Yaskawa INFORM job: X2_34-37(-90,0).JBI

/JOB
//NAME X2_34-37(-90,0)
//POS
///NPOS 361,361,361,9,0,0
///TOOL 0
///POSTYPE PULSE
///PULSE
C00000=-109615,-71844,-36862,18422,13388,2271
C00001=-107008,40287,15446,7646,74688,11911
C00002=-107149,45804,24218,7788,72161,11701
C00003=-108392,48192,28010,10243,72680,1076
C00004=-108392,48392,29954,10302,71604,983
C00005=-108392,48331,29423,10286,71896,1009
C00006=-108010,50265,31522,10186,71551,1114
C00007=-108392,48331,29423,10286,71896,1009
C00008=-108911,49901,30550,10443,72076,8021
C00009=-109414,51873,32709,10619,71831,7821
C00010=-108911,49901,30550,10443,72076,8021
C00011=-102203,43615,23227,8248,72569,10434
C00012=-106081,49085,29485,15378,74997,2308
C00013=-106081,49206,30588,15419,74401,2232
C00014=-106081,49153,30130,15402,74647,2263
C00015=-105730,50968,32108,15326,74307,2347
C00016=-106081,49153,30130,15402,74647,2263
C00017=-108167,43461,21271,12324,74506,6920
C00018=-107374,42085,15448,7738,75637,11845
C00019=-120191,30165,1303,6226,81332,-6626
C00020=-119709,34887,8992,6124,79003,-6581
C00021=-119523,36874,12198,6088,78043,-6565
C00022=-119519,36825,13807,6108,77033,-6613
C00023=-119523,36874,12198,6088,78043,-6565
C00024=-119515,36764,13496,6103,77191,-6604
C00025=-119868,39633,16467,6214,76866,-6741
C00026=-119515,36764,13496,6103,77191,-6604
C00027=-121889,32783,9008,6775,78090,-7366
C00028=-122776,40716,17165,7052,77228,-7717
C00029=-121823,41691,18182,6780,77023,-7402
C00030=-122776,40716,17165,7052,77228,-7717
C00031=-121889,32783,9008,6775,78090,-7366
C00032=-119523,36874,12198,6088,78043,-6565
C00033=-119709,34887,8992,6124,79003,-6581
C00034=-120191,30165,1303,6226,81332,-6626
C00035=-121604,30205,1144,6630,81559,-7083
C00036=-121089,34887,8794,6520,79231,-7034
C00037=-120890,36858,11983,6481,78271,-7017
C00038=-120886,36803,13585,6502,77262,-7069
C00039=-120890,36858,11983,6481,78271,-7017
C00040=-120878,36774,13282,6496,77432,-7057
C00041=-121214,39658,16269,6601,77105,-7189
C00042=-120878,36774,13282,6496,77432,-7057
C00043=-120486,37076,13561,6383,77385,-6926
C00044=-119528,38122,14634,6107,77190,-6608
C00045=-120486,37076,13561,6383,77385,-6926
C00046=-120682,35058,10322,6419,78351,-6942
C00047=-121186,30266,2562,6523,80690,-6990
C00048=-134026,40869,15057,-4047,52311,-47824
C00049=-133273,45805,23219,-4742,49872,-47398
C00050=-132981,47914,26662,-5033,48858,-47219
C00051=-132978,48047,28467,-5116,47820,-47163
C00052=-132981,47914,26662,-5033,48858,-47219
C00053=-132969,48064,28169,-5108,48012,-47169
C00054=-133143,51303,31704,-5016,47492,-47220
C00055=-132969,48064,28169,-5108,48012,-47169
C00056=-135543,46606,26609,-3148,48091,-48321
C00057=-135868,54135,34684,-2953,46980,-48432
C00058=-134925,54643,35244,-3684,46935,-48001
C00059=-135868,54135,34684,-2953,46980,-48432
C00060=-135543,46606,26609,-3148,48091,-48321
C00061=-132981,47914,26662,-5033,48858,-47219
C00062=-133273,45805,23219,-4742,49872,-47398
C00063=-134026,40869,15057,-4047,52311,-47824
C00064=-158164,35728,9631,12841,54320,-57618
C00065=-156933,39530,16487,12369,51918,-57402
C00066=-156452,41160,19364,12190,50934,-57317
C00067=-156450,41229,21096,12367,49926,-57444
C00068=-156452,41160,19364,12190,50934,-57317
C00069=-156479,41102,20610,12346,50159,-57426
C00070=-156356,44237,23924,12335,49721,-57428
C00071=-156479,41102,20610,12346,50159,-57426
C00072=-155785,40986,20547,11858,50036,-57137
C00073=-154785,40646,20189,11137,49940,-56708
C00074=-155785,40986,20547,11858,50036,-57137
C00075=-156262,39303,17617,12037,51024,-57224
C00076=-157483,35375,10637,12509,53434,-57446
C00077=-160593,39475,13550,14508,54241,-58615
C00078=-159342,43270,20469,14089,51785,-58436
C00079=-158853,44905,23381,13934,50776,-58367
C00080=-158852,45007,25149,14138,49770,-58512
C00081=-158853,44905,23381,13934,50776,-58367
C00082=-158854,44932,24718,14094,49990,-58481
C00083=-158703,48121,28150,14084,49505,-58485
C00084=-158854,44932,24718,14094,49990,-58481
C00085=-161444,46441,26342,15939,50249,-59595
C00086=-161040,53766,34331,15923,49060,-59612
C00087=-160097,53171,33669,15238,48978,-59196
C00088=-161040,53766,34331,15923,49060,-59612
C00089=-161444,46441,26342,15939,50249,-59595
C00090=-158853,44905,23381,13934,50776,-58367
C00091=-159342,43270,20469,14089,51785,-58436
C00092=-160593,39475,13550,14508,54241,-58615
C00093=-148971,42504,16746,4915,52183,-53021
C00094=-147979,47046,24523,4355,49683,-52716
C00095=-147593,48996,27807,4132,48646,-52593
C00096=-147590,49137,29621,4197,47605,-52637
C00097=-147593,48996,27807,4132,48646,-52593
C00098=-147610,49163,29309,4198,47810,-52637
C00099=-147661,52475,32942,4273,47281,-52683
C00100=-147610,49163,29309,4198,47810,-52637
C00101=-147454,49128,29272,4080,47808,-52567
C00102=-147457,49325,29466,4083,47790,-52569
C00103=-146486,49526,29681,3347,47716,-52137
C00104=-147457,49325,29466,4083,47790,-52569
C00105=-147454,49128,29272,4080,47808,-52567
C00106=-147593,48996,27807,4132,48646,-52593
C00107=-147979,47046,24523,4355,49683,-52716
C00108=-148753,37651,9035,4624,54413,-52827
C00109=-169007,70240,20067,15770,96475,-54777
C00110=-175404,86334,34832,19373,106938,-55773
C00111=-174173,83341,34513,19133,105400,-55601
C00112=-180960,60737,17059,33421,95392,-55152
C00113=-182232,58952,17300,36312,92073,-55823
C00114=-179527,69319,26237,30671,91177,-56324
C00115=-179117,69620,25739,29739,90864,-56355
C00116=-180097,67994,26330,32410,86483,-57198
C00117=-174100,64042,14056,17976,91926,-56289
C00118=-175447,65123,11808,18399,94042,-56406
C00119=-164161,72,-39985,-6764,90046,-34295
C00120=-130432,-55243,-47386,-13424,82603,8412
C00121=-110572,-56965,-55890,-14658,90278,14468
C00122=-134387,-39172,-38807,12376,86277,-20344
C00123=-136266,-41846,-34601,16059,78566,-27361
C00124=-135424,-39022,-31748,15965,78109,-27121
C00125=-132144,-43884,-34748,15569,76844,-26110
C00126=-133349,-52476,-37829,19150,70304,-22714
C00127=-132707,-53219,-38228,19044,70026,-22517
C00128=-133874,-49344,-36092,21066,73724,-26553
C00129=-127403,-56601,-39797,20204,70737,-24655
C00130=-130575,-58808,-42172,20683,71834,-25657
C00131=-131419,-52897,-41760,13173,72105,-2236
C00132=-151757,-37235,-32664,25855,92713,-16023
C00133=-148694,-31120,-30848,28555,97484,-16481
C00134=-152363,20888,-11521,23566,108052,-25705
C00135=-155491,63274,13853,18429,111086,-34801
C00136=-150514,89045,46229,21307,107758,-32982
C00137=-149106,88504,48693,21100,105732,-32842
C00138=-153882,51041,13508,33623,93530,-12210
C00139=-152694,62068,23397,30426,96150,-11386
C00140=-153686,72545,35966,30292,92124,-9774
C00141=-151360,57639,18849,26215,86885,985
C00142=-146574,44978,5250,17386,80629,11620
C00143=-146389,46654,5686,14273,81867,14897
C00144=-140559,38264,-1160,881,75419,28460
C00145=-140619,46287,2526,1728,82676,28626
C00146=-139837,43342,-3801,1439,85041,28899
C00147=-141798,27002,-27786,2149,91441,28405
C00148=-143772,-19107,-38740,14355,94017,-12677
C00149=-143698,-35148,-33847,20276,92427,-33189
C00150=-141918,-24797,-26817,20326,92921,-32464
C00151=-139594,-23350,-22642,20301,90627,-32011
C00152=-140432,-46735,-33066,23878,71822,-30909
C00153=-143639,-38419,-27501,28411,78321,-12621
C00154=-143508,-41209,-28848,28005,73462,-10092
C00155=-137835,-52557,-35170,23319,62427,898
C00156=-129144,-60406,-38739,13300,52691,14440
C00157=-124267,-62455,-40002,3057,50573,24449
C00158=-118897,-58306,-39599,-7322,55586,36992
C00159=-117935,-60108,-42034,-7672,56240,37337
C00160=-115664,-65010,-47736,-8512,57449,38158
C00161=-121785,-61828,-52329,-5505,69210,35118
C00162=-148930,-33628,-41038,4538,77484,18447
C00163=-163858,24222,1645,10794,81228,7547
C00164=-163712,28964,9442,10824,78886,7392
C00165=-163498,30748,12887,10810,77675,7358
C00166=-163094,25533,8827,6495,74182,-305
C00167=-171402,35198,19720,19438,77476,-19020
C00168=-175083,69400,56807,24741,86302,-36577
C00169=-176478,62304,51821,30230,71876,-61965
C00170=-174700,53660,39403,25265,70725,-61619
C00171=-176244,52382,34806,25393,73168,-61673
C00172=-174832,57379,31343,14926,87681,-59388
C00173=-147451,1111,-29714,5377,100632,-19781
C00174=-112791,-31989,-50015,-2241,90212,24459
C00175=-107981,-35875,-46971,-4517,78040,26268
C00176=-109410,-31915,-41181,-4141,76439,25836
C00177=-109671,-29943,-38250,-4081,75635,25773
C00178=-108634,-25346,-36028,-8315,81190,19632
C00179=-113738,-28838,-38579,-3049,79626,8435
C00180=-120146,-28716,-38356,4151,79685,-1679
C00181=-136605,-12769,-23758,24735,88388,-21929
C00182=-138977,-10728,-20961,25939,84821,-23296
C00183=-136358,-19206,-27135,20431,74888,-32424
C00184=-127631,-24253,-35023,5775,74490,-30240
C00185=-129181,-27934,-40726,6212,76213,-30690
C00186=-139651,-3107,-33687,4364,86662,15844
C00187=-140099,618,-27389,4493,84729,15631
C00188=-140095,1958,-24533,4497,83662,15594
C00189=-138507,5371,-22539,-1336,86874,9491
C00190=-148370,2023,-23416,11466,83880,-10285
C00191=-153111,8749,-17173,17827,86768,-20413
C00192=-156427,18095,-8041,22706,89820,-28931
C00193=-159438,37588,11995,27333,93831,-28775
C00194=-154226,15962,-9104,16757,78816,-38782
C00195=-152712,20066,-9195,12847,84122,-38020
C00196=-154297,18366,-13942,13242,86364,-38311
C00197=-143466,6998,19042,5158,32162,-41222
C00198=-147237,-51968,-50099,-4175,73083,-42408
C00199=3643,-76224,-106676,19950,71810,76872
C00200=6047,-95755,-92046,-14751,98253,9605
C00201=8024,-164446,-133802,-16041,6272,12396
C00202=8024,-164446,-133802,-16041,6272,12396
C00203=80911,-131071,-112390,-19160,57527,-4768
C00204=107387,-112645,-89313,-18613,48039,-3448
C00205=120529,-94925,-67119,-18087,38914,-2179
C00206=102807,-11704,-32462,-5874,76695,-13415
C00207=103436,-3791,-23255,-6127,75148,-13126
C00208=103560,-1765,-20423,-6188,74460,-13051
C00209=103560,-1806,-19122,-6212,73642,-13010
C00210=103601,-1431,-19452,-6214,74041,-13015
C00211=104452,277,-18031,-6506,74110,-12725
C00212=103539,-2063,-20212,-6189,74177,-13043
C00213=120126,-10436,-31938,-6011,80471,6680
C00214=119034,-8056,-29018,-5697,79822,6345
C00215=119034,-8150,-28117,-5707,79221,6375
C00216=119034,-8056,-29018,-5697,79822,6345
C00217=118636,-7203,-28340,-5579,79816,6211
C00218=119064,-5644,-27091,-5704,79877,6351
C00219=118636,-7203,-28340,-5579,79816,6211
C00220=122253,-9472,-30321,-6643,80135,7408
C00221=122707,-3013,-24427,-6779,79866,7571
C00222=122021,-2022,-23613,-6578,79819,7343
C00223=122707,-3013,-24427,-6779,79866,7571
C00224=121204,9301,-16198,-6319,81003,7011
C00225=120979,11415,-12534,-6272,79823,6996
C00226=120979,11346,-11871,-6278,79382,7018
C00227=120979,11415,-12534,-6272,79823,6996
C00228=121673,13624,-10544,-6477,79786,7230
C00229=120979,11415,-12534,-6272,79823,6996
C00230=121039,12182,-11846,-8037,80321,9006
C00231=120294,13253,-10880,-7825,80206,8763
C00232=121039,12182,-11846,-8037,80321,9006
C00233=121310,5674,-20943,-6336,82061,6993
C00234=139815,-25323,-43479,-19,53677,50237
C00235=137572,-18164,-33682,1617,51348,49297
C00236=137572,-18186,-32944,1627,50884,49290
C00237=137572,-18164,-33682,1617,51348,49297
C00238=138000,-16627,-32540,1306,51428,49477
C00239=137572,-18164,-33682,1617,51348,49297
C00240=141541,-18207,-34048,-1274,51544,50959
C00241=141186,-12326,-28968,-1018,51433,50811
C00242=140737,-11536,-28358,-690,51458,50623
C00243=141186,-12326,-28968,-1018,51433,50811
C00244=159686,26179,2441,-14066,53601,58348
C00245=159232,27229,5186,-13963,52408,58323
C00246=159232,27222,5932,-14048,51958,58386
C00247=159232,27229,5186,-13963,52408,58323
C00248=159232,27225,5485,-13997,52227,58349
C00249=159220,29212,7438,-14024,52052,58369
C00250=159232,27225,5485,-13997,52227,58349
C00251=164735,35698,13654,-29808,58437,68077
C00252=164028,35618,13572,-29436,58200,67836
C00253=164735,35698,13654,-29808,58437,68077
C00254=161795,29787,7764,-15728,52595,59373
C00255=161795,29788,8601,-15834,52098,59452
C00256=161795,29787,7764,-15728,52595,59373
C00257=161783,31729,9695,-15761,52409,59396
C00258=161795,29787,7764,-15728,52595,59373
C00259=165243,28841,7606,-18106,52930,60800
C00260=165806,38731,16984,-22046,53706,63214
C00261=165192,38605,16853,-21659,53559,62976
C00262=165806,38731,16984,-22046,53706,63214
C00263=161708,46386,23154,-8907,61269,44547
C00264=161224,48066,26131,-8737,60259,44442
C00265=161222,48202,27939,-8826,59228,44523
C00266=161224,48066,26131,-8737,60259,44442
C00267=161238,48238,27638,-8816,59431,44513
C00268=161118,51495,31180,-8798,58918,44508
C00269=161238,48238,27638,-8816,59431,44513
C00270=161086,48113,27502,-8735,59433,44454
C00271=161078,48307,27691,-8732,59416,44452
C00272=160108,47930,27281,-8216,59373,44078
C00273=161078,48307,27691,-8732,59416,44452
C00274=161086,48113,27502,-8735,59433,44454
C00275=161224,48066,26131,-8737,60259,44442
C00276=161708,46386,23154,-8907,61269,44547
C00277=162944,42495,16096,-9351,63722,44812
C00278=174609,85782,55206,-18480,94121,57514
C00279=173388,84153,56528,-18357,92279,57362
C00280=178295,72858,49572,-29598,87914,53870
C00281=178363,71681,49458,-30316,81279,55416
C00282=178775,74747,53745,-31442,79609,55982
C00283=178120,80280,53499,-25679,87195,54196
C00284=177788,66292,45128,-22799,80541,57078
C00285=165876,20944,-7359,-14016,91072,47752
C00286=144031,-8096,-47002,481,102749,33013
C00287=113249,-55125,-55779,6617,87879,-14622
C00288=105402,-49476,-43093,17129,78821,-17705
C00289=107372,-45114,-37354,16923,77172,-17229
C00290=107897,-43226,-34630,16890,76385,-17150
C00291=123036,-54169,-41018,-3647,66196,-9526
C00292=125103,-54109,-40569,-7539,65613,-9158
C00293=133018,-52183,-38196,-18552,67287,-3963
C00294=135096,-56008,-41994,-19101,68310,-3149
C00295=148619,-36280,-33179,-26254,90102,11601
C00296=132022,-46525,-51369,-8915,93592,12104
C00297=152394,4325,-31091,-21424,100011,27739
C00298=150620,74441,30669,-21497,109248,32750
C00299=152126,53419,9650,-25324,101365,34081
C00300=152823,56464,14992,-29675,98105,11003
C00301=153512,66710,26766,-28901,94570,8735
C00302=151176,53481,12027,-24882,88967,-903
C00303=148217,46273,4019,-19056,85273,-8690
C00304=145575,40234,-2364,-10924,81880,-17637
C00305=142774,42237,-1321,-4504,82417,-25550
C00306=141310,41249,-3509,-1904,83312,-28397
C00307=140520,38377,-9680,-1608,85617,-28672
C00308=145482,-30493,-50756,-14636,95383,13188
C00309=142176,-26033,-28146,-20229,92686,32606
C00310=139838,-24569,-23969,-20194,90398,32145
C00311=141333,-43488,-32424,-24355,75177,35516
C00312=142946,-39788,-29545,-27566,77515,12382
C00313=142712,-38988,-29426,-26650,76094,9122
C00314=137490,-51139,-36024,-22440,64589,-1384
C00315=129219,-61272,-40095,-12800,52551,-14455
C00316=125098,-62268,-41395,-3949,52110,-22670
C00317=120434,-59895,-41306,5152,54802,-34175
C00318=118218,-60267,-42467,7826,55944,-37248
C00319=115940,-65207,-48159,8687,57132,-38075
C00320=158051,-33814,-49892,-7441,80913,-13725
C00321=163513,25616,3177,-10792,80459,-7597
C00322=163372,30455,11081,-10830,78103,-7439
C00323=163993,28142,11085,-12803,74423,-6981
C00324=161648,29238,11147,-4496,75447,-179
C00325=171143,45412,28292,-19077,81279,23270
C00326=173705,65046,50293,-22854,85176,36170
C00327=173974,62485,49606,-24076,73199,49227
C00328=172570,70781,55370,-19160,78152,47867
C00329=174025,68948,50025,-19270,80716,47984
C00330=170072,38309,9009,-5458,81396,48416
C00331=145937,-33300,-50613,-2555,87892,10434
C00332=117969,-26674,-50251,1455,96093,-22658
C00333=108065,-36096,-47601,4778,77881,-26213
C00334=109507,-32110,-41823,4391,76297,-25779
C00335=109013,-37865,-42571,5415,69231,-26193
C00336=107679,-33877,-40967,9851,74714,-20356
C00337=113110,-32097,-41032,3661,77261,-8676
C00338=119719,-29513,-40298,-3828,79988,1546
C00339=130402,-22376,-34110,-15555,82843,20591
C00340=132503,-6978,-23545,-15597,88653,21115
C00341=133170,-4219,-21374,-15691,88857,21320
C00342=127848,-25408,-36231,-5685,74178,30350
C00343=129407,-29126,-41925,-6135,75876,30806
C00344=139811,-3516,-34603,-4319,86523,-15767
C00345=140259,233,-28314,-4452,84609,-15556
C00346=139695,2013,-26001,-4296,84073,-15716
C00347=138357,5152,-24179,1260,87195,-9766
C00348=142581,5884,-23661,-3711,87904,1101
C00349=150814,13438,-16434,-14780,91136,16214
C00350=153585,30594,-714,-18230,97958,27100
C00351=154794,42503,11376,-18274,96962,27667
C00352=154809,42525,11398,-18275,96963,27672
C00353=153093,18834,-10833,-12947,84050,38162
C00354=154693,17143,-15552,-13354,86281,38457
C00355=149017,-30265,-44675,-21897,62232,30468
C00356=102406,-109115,-77602,-2898,35707,-11807
C00357=80911,-131071,-112390,-19160,57527,-4768
C00358=8024,-164446,-133802,-16041,6272,12396
C00359=8024,-164446,-133802,-16041,6272,12396
C00360=1579,-114561,-88072,141,60969,-160
BC00000=287767,672594,392898
BC00001=287767,702390,199743
BC00002=287767,702390,199743
BC00003=287767,702390,199743
BC00004=287767,702390,199743
BC00005=287767,702390,199743
BC00006=287767,702390,199743
BC00007=287767,702390,199743
BC00008=287767,702390,199743
BC00009=287767,702390,199743
BC00010=287767,702390,199743
BC00011=287767,702390,199743
BC00012=287767,702390,199743
BC00013=287767,702390,199743
BC00014=287767,702390,199743
BC00015=287767,702390,199743
BC00016=287767,702390,199743
BC00017=287767,702390,199743
BC00018=287767,702390,199743
BC00019=325466,709124,183073
BC00020=325466,709124,183073
BC00021=325466,709124,183073
BC00022=325466,709124,183073
BC00023=325466,709124,183073
BC00024=325466,709124,183073
BC00025=325466,709124,183073
BC00026=325466,709124,183073
BC00027=325466,709124,183073
BC00028=325466,709124,183073
BC00029=325466,709124,183073
BC00030=325466,709124,183073
BC00031=325466,709124,183073
BC00032=325466,709124,183073
BC00033=325466,709124,183073
BC00034=325466,709124,183073
BC00035=304409,729721,181352
BC00036=304409,729721,181352
BC00037=304409,729721,181352
BC00038=304409,729721,181352
BC00039=304409,729721,181352
BC00040=304409,729721,181352
BC00041=304409,729721,181352
BC00042=304409,729721,181352
BC00043=304409,729721,181352
BC00044=304409,729721,181352
BC00045=304409,729721,181352
BC00046=304409,729721,181352
BC00047=304409,729721,181352
BC00048=360941,686135,119054
BC00049=360941,686135,119054
BC00050=360941,686135,119054
BC00051=360941,686135,119054
BC00052=360941,686135,119054
BC00053=360941,686135,119054
BC00054=360941,686135,119054
BC00055=360941,686135,119054
BC00056=360941,686135,119054
BC00057=360941,686135,119054
BC00058=360941,686135,119054
BC00059=360941,686135,119054
BC00060=360941,686135,119054
BC00061=360941,686135,119054
BC00062=360941,686135,119054
BC00063=360941,686135,119054
BC00064=398174,742009,118025
BC00065=398174,742009,118025
BC00066=398174,742009,118025
BC00067=398174,742009,118025
BC00068=398174,742009,118025
BC00069=398174,742009,118025
BC00070=398174,742009,118025
BC00071=398174,742009,118025
BC00072=398174,742009,118025
BC00073=398174,742009,118025
BC00074=398174,742009,118025
BC00075=398174,742009,118025
BC00076=398174,742009,118025
BC00077=397434,738268,118311
BC00078=397434,738268,118311
BC00079=397434,738268,118311
BC00080=397434,738268,118311
BC00081=397434,738268,118311
BC00082=397434,738268,118311
BC00083=397434,738268,118311
BC00084=397434,738268,118311
BC00085=397434,738268,118311
BC00086=397434,738268,118311
BC00087=397434,738268,118311
BC00088=397434,738268,118311
BC00089=397434,738268,118311
BC00090=397434,738268,118311
BC00091=397434,738268,118311
BC00092=397434,738268,118311
BC00093=337757,747913,121043
BC00094=337757,747913,121043
BC00095=337757,747913,121043
BC00096=337757,747913,121043
BC00097=337757,747913,121043
BC00098=337757,747913,121043
BC00099=337757,747913,121043
BC00100=337757,747913,121043
BC00101=337757,747913,121043
BC00102=337757,747913,121043
BC00103=337757,747913,121043
BC00104=337757,747913,121043
BC00105=337757,747913,121043
BC00106=337757,747913,121043
BC00107=337757,747913,121043
BC00108=337757,747913,121043
BC00109=382499,793323,31443
BC00110=398174,809232,53
BC00111=398174,809232,53
BC00112=398174,809232,53
BC00113=398174,809232,53
BC00114=398174,809232,53
BC00115=398174,809232,53
BC00116=398174,809232,53
BC00117=398174,809232,53
BC00118=398174,809232,53
BC00119=378399,812249,125880
BC00120=350148,816882,305631
BC00121=350148,816882,305631
BC00122=350717,816957,305463
BC00123=350717,816957,305463
BC00124=350717,816957,305463
BC00125=350717,816957,305463
BC00126=350717,816957,305459
BC00127=350717,816957,305459
BC00128=350717,816957,305459
BC00129=350717,816957,305459
BC00130=350717,816957,305459
BC00131=350717,816957,305463
BC00132=350717,816957,305463
BC00133=350148,816882,305631
BC00134=357486,783574,171223
BC00135=363745,755164,56581
BC00136=350108,749289,42117
BC00137=350108,749289,42117
BC00138=350108,749289,42117
BC00139=350108,749289,42117
BC00140=350108,749289,42117
BC00141=350108,749289,42117
BC00142=350108,749289,42117
BC00143=350108,749289,42117
BC00144=350108,749289,42117
BC00145=350108,749289,42117
BC00146=350108,749289,42117
BC00147=350045,748919,44151
BC00148=332829,802151,218589
BC00149=324221,828766,305808
BC00150=324283,829135,303773
BC00151=324283,829135,303773
BC00152=324283,829135,303773
BC00153=324283,829135,303773
BC00154=324283,829135,303773
BC00155=324283,829135,303773
BC00156=324283,829135,303773
BC00157=324283,829135,303773
BC00158=324283,829135,303773
BC00159=324283,829135,303773
BC00160=324283,829135,303773
BC00161=324221,828766,305808
BC00162=365904,809152,256676
BC00163=398174,795215,220015
BC00164=398174,795215,220015
BC00165=398174,795215,220015
BC00166=398174,795215,220015
BC00167=398174,795215,220015
BC00168=398174,795215,220015
BC00169=398174,795215,220015
BC00170=398174,795215,220015
BC00171=398174,795215,220015
BC00172=398174,795215,220015
BC00173=365121,791381,219974
BC00174=328869,787176,219929
BC00175=328869,787176,219929
BC00176=328869,787176,219929
BC00177=328869,787176,219929
BC00178=328869,787176,219929
BC00179=328869,787176,219929
BC00180=328869,787176,219929
BC00181=328869,787176,219929
BC00182=328869,787176,219929
BC00183=328869,787176,219929
BC00184=328869,787176,219929
BC00185=328869,787176,219929
BC00186=366743,775181,149862
BC00187=366743,775181,149862
BC00188=366743,775181,149862
BC00189=366743,775181,149862
BC00190=366743,775181,149862
BC00191=366743,775181,149862
BC00192=366743,775181,149862
BC00193=366743,775181,149862
BC00194=366743,775181,149862
BC00195=366743,775181,149862
BC00196=366743,775181,149862
BC00197=366743,675039,355777
BC00198=366743,675039,355777
BC00199=199464,674570,1075173
BC00200=95044,675039,919146
BC00201=95044,675039,1075229
BC00202=235813,1345575,1075229
BC00203=291733,1363613,501241
BC00204=295042,1365829,344881
BC00205=288108,1367960,194507
BC00206=288108,1365832,194507
BC00207=288108,1369193,194507
BC00208=288108,1369264,194507
BC00209=288108,1369264,194507
BC00210=288108,1369614,194507
BC00211=288108,1369614,194507
BC00212=288108,1368913,194507
BC00213=325834,1368698,177132
BC00214=325834,1367902,177132
BC00215=325834,1367902,177132
BC00216=325834,1367902,177132
BC00217=325834,1367902,177132
BC00218=325834,1367902,177132
BC00219=325834,1367902,177132
BC00220=325834,1368223,177132
BC00221=325834,1368768,177132
BC00222=325834,1368768,177132
BC00223=325834,1368768,177132
BC00224=304798,1367887,175873
BC00225=304798,1368278,175873
BC00226=304798,1368278,175873
BC00227=304798,1368278,175873
BC00228=304798,1368278,175873
BC00229=304798,1368278,175873
BC00230=304798,1368278,175873
BC00231=304798,1368278,175873
BC00232=304798,1368278,175873
BC00233=304798,1368714,175873
BC00234=360316,1368040,111260
BC00235=360316,1367747,111260
BC00236=360316,1367747,111260
BC00237=360316,1367747,111260
BC00238=360316,1367747,111260
BC00239=360316,1367747,111260
BC00240=360316,1368265,111260
BC00241=360316,1367537,111260
BC00242=360316,1367537,111260
BC00243=360316,1367537,111260
BC00244=398174,1367762,110837
BC00245=398174,1365917,110837
BC00246=398174,1365917,110837
BC00247=398174,1365917,110837
BC00248=398174,1365917,110837
BC00249=398174,1365917,110837
BC00250=398174,1365917,110837
BC00251=398174,1365917,110837
BC00252=398174,1365917,110837
BC00253=398174,1365917,110837
BC00254=397184,1368437,111272
BC00255=397184,1368437,111272
BC00256=397184,1368437,111272
BC00257=397184,1368437,111272
BC00258=397184,1368437,111272
BC00259=397184,1366459,111272
BC00260=397184,1367282,111272
BC00261=397184,1367282,111272
BC00262=397184,1367282,111272
BC00263=375501,1345864,156348
BC00264=375501,1345864,156348
BC00265=375501,1345864,156348
BC00266=375501,1345864,156348
BC00267=375501,1345864,156348
BC00268=375501,1345864,156348
BC00269=375501,1345864,156348
BC00270=375501,1345864,156348
BC00271=375501,1345864,156348
BC00272=375501,1345864,156348
BC00273=375501,1345864,156348
BC00274=375501,1345864,156348
BC00275=375501,1345864,156348
BC00276=375501,1345864,156348
BC00277=375501,1345864,156348
BC00278=398174,1321783,135113
BC00279=398174,1321783,135113
BC00280=398174,1321783,135113
BC00281=398174,1321783,135113
BC00282=398174,1321783,135113
BC00283=398174,1321783,135110
BC00284=398174,1321783,199558
BC00285=369955,1320476,190565
BC00286=332653,1318400,176274
BC00287=350446,1306885,300644
BC00288=351050,1306811,300466
BC00289=351050,1306811,300466
BC00290=351050,1306811,300466
BC00291=351050,1306811,300466
BC00292=351050,1306811,300466
BC00293=351050,1306811,300466
BC00294=351050,1306811,300466
BC00295=351050,1306811,300466
BC00296=350446,1306885,300644
BC00297=350330,1345569,140511
BC00298=350318,1362954,38397
BC00299=350319,1362252,38395
BC00300=350318,1369188,38397
BC00301=350318,1369188,38397
BC00302=350318,1369188,38397
BC00303=350318,1369188,38393
BC00304=350318,1369188,38397
BC00305=350318,1369188,38397
BC00306=350318,1369188,38397
BC00307=350318,1369188,38397
BC00308=332907,1319511,215580
BC00309=324469,1294535,299337
BC00310=324469,1294535,299337
BC00311=324469,1294535,299337
BC00312=324469,1294535,299337
BC00313=324469,1294535,299337
BC00314=324469,1294535,299337
BC00315=324469,1294535,299337
BC00316=324469,1294535,299337
BC00317=324470,1294536,299336
BC00318=324469,1294535,299337
BC00319=324469,1294535,299337
BC00320=378057,1319426,238838
BC00321=398174,1331142,220624
BC00322=398174,1331142,220624
BC00323=398174,1331142,220624
BC00324=398174,1331142,220624
BC00325=398174,1331142,220624
BC00326=398174,1331142,220624
BC00327=398174,1331142,220624
BC00328=398174,1331142,220624
BC00329=398174,1331142,220624
BC00330=398174,1328620,215389
BC00331=359686,1333158,214696
BC00332=329122,1336762,214146
BC00333=329122,1336762,214146
BC00334=329122,1336762,214146
BC00335=329122,1336762,214146
BC00336=329122,1336762,214146
BC00337=329122,1336762,214146
BC00338=329122,1336762,214146
BC00339=329122,1336762,214146
BC00340=329122,1336762,214146
BC00341=329122,1336762,214146
BC00342=329122,1336762,214146
BC00343=329122,1336762,214146
BC00344=367015,1348719,144696
BC00345=367015,1348719,144696
BC00346=367015,1348719,144696
BC00347=367015,1348719,144696
BC00348=367015,1348719,144696
BC00349=367015,1348719,144696
BC00350=367015,1348719,144696
BC00351=367015,1348719,144696
BC00352=367015,1348719,144696
BC00353=367015,1348719,144696
BC00354=367015,1348719,144696
BC00355=346608,1354830,157578
BC00356=288108,1360159,194507
BC00357=269895,1363613,501241
BC00358=235813,1345575,1075229
BC00359=95044,675039,1075229
BC00360=127053,672594,1075229
EC00000=-798156,0
EC00001=-798156,0
EC00002=-798156,0
EC00003=-798156,0
EC00004=-798156,0
EC00005=-798156,0
EC00006=-798156,0
EC00007=-798156,0
EC00008=-798156,0
EC00009=-798156,0
EC00010=-798156,0
EC00011=-798156,0
EC00012=-798156,0
EC00013=-798156,0
EC00014=-798156,0
EC00015=-798156,0
EC00016=-798156,0
EC00017=-798156,0
EC00018=-798156,0
EC00019=-798156,0
EC00020=-798156,0
EC00021=-798156,0
EC00022=-798156,0
EC00023=-798156,0
EC00024=-798156,0
EC00025=-798156,0
EC00026=-798156,0
EC00027=-798156,0
EC00028=-798156,0
EC00029=-798156,0
EC00030=-798156,0
EC00031=-798156,0
EC00032=-798156,0
EC00033=-798156,0
EC00034=-798156,0
EC00035=-798156,0
EC00036=-798156,0
EC00037=-798156,0
EC00038=-798156,0
EC00039=-798156,0
EC00040=-798156,0
EC00041=-798156,0
EC00042=-798156,0
EC00043=-798156,0
EC00044=-798156,0
EC00045=-798156,0
EC00046=-798156,0
EC00047=-798156,0
EC00048=-798156,0
EC00049=-798156,0
EC00050=-798156,0
EC00051=-798156,0
EC00052=-798156,0
EC00053=-798156,0
EC00054=-798156,0
EC00055=-798156,0
EC00056=-798156,0
EC00057=-798156,0
EC00058=-798156,0
EC00059=-798156,0
EC00060=-798156,0
EC00061=-798156,0
EC00062=-798156,0
EC00063=-798156,0
EC00064=-798156,0
EC00065=-798156,0
EC00066=-798156,0
EC00067=-798156,0
EC00068=-798156,0
EC00069=-798156,0
EC00070=-798156,0
EC00071=-798156,0
EC00072=-798156,0
EC00073=-798156,0
EC00074=-798156,0
EC00075=-798156,0
EC00076=-798156,0
EC00077=-798156,0
EC00078=-798156,0
EC00079=-798156,0
EC00080=-798156,0
EC00081=-798156,0
EC00082=-798156,0
EC00083=-798156,0
EC00084=-798156,0
EC00085=-798156,0
EC00086=-798156,0
EC00087=-798156,0
EC00088=-798156,0
EC00089=-798156,0
EC00090=-798156,0
EC00091=-798156,0
EC00092=-798156,0
EC00093=-798156,0
EC00094=-798156,0
EC00095=-798156,0
EC00096=-798156,0
EC00097=-798156,0
EC00098=-798156,0
EC00099=-798156,0
EC00100=-798156,0
EC00101=-798156,0
EC00102=-798156,0
EC00103=-798156,0
EC00104=-798156,0
EC00105=-798156,0
EC00106=-798156,0
EC00107=-798156,0
EC00108=-798156,0
EC00109=-798156,0
EC00110=-798156,0
EC00111=-798156,0
EC00112=-798156,0
EC00113=-798156,0
EC00114=-798156,0
EC00115=-798156,0
EC00116=-798156,0
EC00117=-798156,0
EC00118=-798156,0
EC00119=-798156,0
EC00120=-798156,0
EC00121=-798156,0
EC00122=-798156,0
EC00123=-798156,0
EC00124=-798156,0
EC00125=-798156,0
EC00126=-798155,0
EC00127=-798155,0
EC00128=-798155,0
EC00129=-798155,0
EC00130=-798155,0
EC00131=-798156,0
EC00132=-798156,0
EC00133=-798156,0
EC00134=-798156,0
EC00135=-798156,0
EC00136=-798156,0
EC00137=-798156,0
EC00138=-798156,0
EC00139=-798156,0
EC00140=-798156,0
EC00141=-798156,0
EC00142=-798156,0
EC00143=-798156,0
EC00144=-798156,0
EC00145=-798156,0
EC00146=-798156,0
EC00147=-798156,0
EC00148=-798156,0
EC00149=-798156,0
EC00150=-798156,0
EC00151=-798156,0
EC00152=-798156,0
EC00153=-798156,0
EC00154=-798156,0
EC00155=-798156,0
EC00156=-798156,0
EC00157=-798156,0
EC00158=-798156,0
EC00159=-798156,0
EC00160=-798156,0
EC00161=-798156,0
EC00162=-798156,0
EC00163=-798156,0
EC00164=-798156,0
EC00165=-798156,0
EC00166=-798156,0
EC00167=-798156,0
EC00168=-798156,0
EC00169=-798156,0
EC00170=-798156,0
EC00171=-798156,0
EC00172=-798156,0
EC00173=-798156,0
EC00174=-798156,0
EC00175=-798156,0
EC00176=-798156,0
EC00177=-798156,0
EC00178=-798156,0
EC00179=-798156,0
EC00180=-798156,0
EC00181=-798156,0
EC00182=-798156,0
EC00183=-798156,0
EC00184=-798156,0
EC00185=-798156,0
EC00186=-798156,0
EC00187=-798156,0
EC00188=-798156,0
EC00189=-798156,0
EC00190=-798156,0
EC00191=-798156,0
EC00192=-798156,0
EC00193=-798156,0
EC00194=-798156,0
EC00195=-798156,0
EC00196=-798156,0
EC00197=-798156,0
EC00198=-798156,0
EC00199=-798156,0
EC00200=-798156,0
EC00201=798156,0
EC00202=798156,0
EC00203=798156,0
EC00204=798156,0
EC00205=798156,0
EC00206=798156,0
EC00207=798156,0
EC00208=798156,0
EC00209=798156,0
EC00210=798156,0
EC00211=798156,0
EC00212=798156,0
EC00213=798156,0
EC00214=798156,0
EC00215=798156,0
EC00216=798156,0
EC00217=798156,0
EC00218=798156,0
EC00219=798156,0
EC00220=798156,0
EC00221=798156,0
EC00222=798156,0
EC00223=798156,0
EC00224=798156,0
EC00225=798156,0
EC00226=798156,0
EC00227=798156,0
EC00228=798156,0
EC00229=798156,0
EC00230=798156,0
EC00231=798156,0
EC00232=798156,0
EC00233=798156,0
EC00234=798156,0
EC00235=798156,0
EC00236=798156,0
EC00237=798156,0
EC00238=798156,0
EC00239=798156,0
EC00240=798156,0
EC00241=798156,0
EC00242=798156,0
EC00243=798156,0
EC00244=798156,0
EC00245=798156,0
EC00246=798156,0
EC00247=798156,0
EC00248=798156,0
EC00249=798156,0
EC00250=798156,0
EC00251=798156,0
EC00252=798156,0
EC00253=798156,0
EC00254=798156,0
EC00255=798156,0
EC00256=798156,0
EC00257=798156,0
EC00258=798156,0
EC00259=798156,0
EC00260=798156,0
EC00261=798156,0
EC00262=798156,0
EC00263=798156,0
EC00264=798156,0
EC00265=798156,0
EC00266=798156,0
EC00267=798156,0
EC00268=798156,0
EC00269=798156,0
EC00270=798156,0
EC00271=798156,0
EC00272=798156,0
EC00273=798156,0
EC00274=798156,0
EC00275=798156,0
EC00276=798156,0
EC00277=798156,0
EC00278=798156,0
EC00279=798156,0
EC00280=798156,0
EC00281=798156,0
EC00282=798156,0
EC00283=798155,1
EC00284=798155,1
EC00285=798155,1
EC00286=798156,0
EC00287=798156,0
EC00288=798156,0
EC00289=798156,0
EC00290=798156,0
EC00291=798156,0
EC00292=798156,0
EC00293=798156,0
EC00294=798156,0
EC00295=798156,0
EC00296=798156,0
EC00297=798156,0
EC00298=798156,0
EC00299=798155,0
EC00300=798156,0
EC00301=798156,0
EC00302=798156,0
EC00303=798155,1
EC00304=798156,0
EC00305=798156,0
EC00306=798156,0
EC00307=798156,0
EC00308=798156,0
EC00309=798156,0
EC00310=798156,0
EC00311=798156,0
EC00312=798156,0
EC00313=798156,0
EC00314=798156,0
EC00315=798156,0
EC00316=798156,0
EC00317=798155,1
EC00318=798156,0
EC00319=798156,0
EC00320=798156,0
EC00321=798156,0
EC00322=798156,0
EC00323=798156,0
EC00324=798156,0
EC00325=798156,0
EC00326=798156,0
EC00327=798156,0
EC00328=798156,0
EC00329=798156,0
EC00330=798156,0
EC00331=798156,0
EC00332=798156,0
EC00333=798156,0
EC00334=798156,0
EC00335=798156,0
EC00336=798156,0
EC00337=798156,0
EC00338=798156,0
EC00339=798156,0
EC00340=798156,0
EC00341=798156,0
EC00342=798156,0
EC00343=798156,0
EC00344=798156,0
EC00345=798156,0
EC00346=798156,0
EC00347=798156,0
EC00348=798156,0
EC00349=798156,0
EC00350=798156,0
EC00351=798156,0
EC00352=798156,0
EC00353=798156,0
EC00354=798156,0
EC00355=798156,0
EC00356=798156,0
EC00357=798156,0
EC00358=798156,0
EC00359=798156,0
EC00360=798156,0
///POSTYPE BASE
///RECTAN
///RCONF 0,0,0,0,0,0,0,0,0,0,0,0,0,0,0,0,0,0,0,0,0,0,0,0
P00006=0.222,-3.123,-1.508,0.0000,0.0000,0.0000
P00021=-0.225,-6.128,-0.405,0.0000,0.0000,0.0000
P00022=0.222,-3.123,-1.508,0.0000,0.0000,0.0000
P00023=0.143,-0.036,0.682,0.0000,0.0000,0.0000
P00024=0.145,-0.552,1.326,0.0000,0.0000,0.0000
P00025=-2.003,0.006,0.728,0.0000,0.0000,0.0000
P00026=0.562,-0.002,-0.337,0.0000,0.0000,0.0000
P00027=-0.746,0.015,-9.096,0.0000,0.0000,0.0000
P00031=1.853,-0.001,-1.549,0.0000,0.0000,0.0000
//INST
///DATE 2024/04/08 11:51
///ATTR SC,RW
///GROUP1 RB1,BS1
///GROUP2 ST1
NOP
'X2_34-37(-90,0)
'210,0
MOVJ C00000 BC00000 VJ=100.00  +MOVJ EC00000 VJ=100.00
'Path S3633
SFTOF3D
MOVJ C00001 BC00001 VJ=100.00  +MOVJ EC00001 VJ=100.00
MOVL C00002 BC00002 V=800.0  +MOVJ EC00002 VJ=100.00
SMOVL C00003 BC00003 V=166.7  +MOVJ EC00003
SREFP 3 C00004 BC00004  +REFP EC00004
CALL JOB:SEARCH-R1-S13D
SET P021 P006
SFTON3D P021
SMOVL C00005 BC00005 V=166.7  +MOVJ EC00005
SREFP 3 C00006 BC00006  +REFP EC00006
CALL JOB:SEARCH-R1-S13D
SET P021 P006
SFTON3D P021
SMOVL C00007 BC00007 V=166.7  +MOVJ EC00007
SMOVL C00008 BC00008 V=166.7  +MOVJ EC00008
SREFP 3 C00009 BC00009  +REFP EC00009
CALL JOB:SEARCH-R1-S13D
SET P021 P006
SFTON3D P021
SMOVL C00010 BC00010 V=166.7  +MOVJ EC00010
SFTOF3D
SMOVL C00011 BC00011 V=250.0  +MOVJ EC00011
SMOVL C00012 BC00012 V=166.7  +MOVJ EC00012
SREFP 3 C00013 BC00013  +REFP EC00013
CALL JOB:SEARCH-R1-S13D
SET P031 P006
SFTON3D P031
SMOVL C00014 BC00014 V=166.7  +MOVJ EC00014
SREFP 3 C00015 BC00015  +REFP EC00015
CALL JOB:SEARCH-R1-S13D
SET P031 P006
SFTON3D P031
SMOVL C00016 BC00016 V=166.7  +MOVJ EC00016
MOVL C00017 BC00017 V=800.0  +MOVJ EC00017 VJ=100.00
MOVL C00018 BC00018 V=1000.0  +MOVJ EC00018 VJ=100.00
'EndPath S3633
'Path S4258
SFTOF3D
MOVJ C00019 BC00019 VJ=100.00  +MOVJ EC00019 VJ=100.00
MOVL C00020 BC00020 V=800.0  +MOVJ EC00020 VJ=100.00
SMOVL C00021 BC00021 V=166.7  +MOVJ EC00021
SREFP 3 C00022 BC00022  +REFP EC00022
CALL JOB:SEARCH-R1-S13D
SET P022 P006
SFTON3D P022
SMOVL C00023 BC00023 V=166.7  +MOVJ EC00023
SMOVL C00024 BC00024 V=166.7  +MOVJ EC00024
SREFP 3 C00025 BC00025  +REFP EC00025
CALL JOB:SEARCH-R1-S13D
SET P022 P006
SFTON3D P022
SMOVL C00026 BC00026 V=166.7  +MOVJ EC00026
SMOVL C00027 BC00027 V=166.7  +MOVJ EC00027
SMOVL C00028 BC00028 V=166.7  +MOVJ EC00028
SREFP 3 C00029 BC00029  +REFP EC00029
CALL JOB:SEARCH-R1-S13D
SET P022 P006
SFTON3D P022
SMOVL C00030 BC00030 V=166.7  +MOVJ EC00030
SMOVL C00031 BC00031 V=166.7  +MOVJ EC00031
SMOVL C00032 BC00032 V=166.7  +MOVJ EC00032
MOVL C00033 BC00033 V=800.0  +MOVJ EC00033 VJ=100.00
MOVL C00034 BC00034 V=1000.0  +MOVJ EC00034 VJ=100.00
'EndPath S4258
'Path S4259
SFTOF3D
MOVJ C00035 BC00035 VJ=100.00  +MOVJ EC00035 VJ=100.00
MOVL C00036 BC00036 V=800.0  +MOVJ EC00036 VJ=100.00
SMOVL C00037 BC00037 V=166.7  +MOVJ EC00037
SREFP 3 C00038 BC00038  +REFP EC00038
CALL JOB:SEARCH-R1-S13D
SET P023 P006
SFTON3D P023
SMOVL C00039 BC00039 V=166.7  +MOVJ EC00039
SMOVL C00040 BC00040 V=166.7  +MOVJ EC00040
SREFP 3 C00041 BC00041  +REFP EC00041
CALL JOB:SEARCH-R1-S13D
SET P023 P006
SFTON3D P023
SMOVL C00042 BC00042 V=166.7  +MOVJ EC00042
SMOVL C00043 BC00043 V=166.7  +MOVJ EC00043
SREFP 3 C00044 BC00044  +REFP EC00044
CALL JOB:SEARCH-R1-S13D
SET P023 P006
SFTON3D P023
SMOVL C00045 BC00045 V=166.7  +MOVJ EC00045
MOVL C00046 BC00046 V=800.0  +MOVJ EC00046 VJ=100.00
MOVL C00047 BC00047 V=1000.0  +MOVJ EC00047 VJ=100.00
'EndPath S4259
'Path S4260
SFTOF3D
MOVJ C00048 BC00048 VJ=100.00  +MOVJ EC00048 VJ=100.00
MOVL C00049 BC00049 V=800.0  +MOVJ EC00049 VJ=100.00
SMOVL C00050 BC00050 V=166.7  +MOVJ EC00050
SREFP 3 C00051 BC00051  +REFP EC00051
CALL JOB:SEARCH-R1-S13D
SET P024 P006
SFTON3D P024
SMOVL C00052 BC00052 V=166.7  +MOVJ EC00052
SMOVL C00053 BC00053 V=166.7  +MOVJ EC00053
SREFP 3 C00054 BC00054  +REFP EC00054
CALL JOB:SEARCH-R1-S13D
SET P024 P006
SFTON3D P024
SMOVL C00055 BC00055 V=166.7  +MOVJ EC00055
SMOVL C00056 BC00056 V=166.7  +MOVJ EC00056
SMOVL C00057 BC00057 V=166.7  +MOVJ EC00057
SREFP 3 C00058 BC00058  +REFP EC00058
CALL JOB:SEARCH-R1-S13D
SET P024 P006
SFTON3D P024
SMOVL C00059 BC00059 V=166.7  +MOVJ EC00059
SMOVL C00060 BC00060 V=166.7  +MOVJ EC00060
SMOVL C00061 BC00061 V=166.7  +MOVJ EC00061
MOVL C00062 BC00062 V=800.0  +MOVJ EC00062 VJ=100.00
MOVL C00063 BC00063 V=1000.0  +MOVJ EC00063 VJ=100.00
'EndPath S4260
'Path S4261
SFTOF3D
MOVJ C00064 BC00064 VJ=100.00  +MOVJ EC00064 VJ=100.00
MOVL C00065 BC00065 V=800.0  +MOVJ EC00065 VJ=100.00
SMOVL C00066 BC00066 V=166.7  +MOVJ EC00066
SREFP 3 C00067 BC00067  +REFP EC00067
CALL JOB:SEARCH-R1-S13D
SET P025 P006
SFTON3D P025
SMOVL C00068 BC00068 V=166.7  +MOVJ EC00068
SMOVL C00069 BC00069 V=166.7  +MOVJ EC00069
SREFP 3 C00070 BC00070  +REFP EC00070
CALL JOB:SEARCH-R1-S13D
SET P025 P006
SFTON3D P025
SMOVL C00071 BC00071 V=166.7  +MOVJ EC00071
SMOVL C00072 BC00072 V=166.7  +MOVJ EC00072
SREFP 3 C00073 BC00073  +REFP EC00073
CALL JOB:SEARCH-R1-S13D
SET P025 P006
SFTON3D P025
SMOVL C00074 BC00074 V=166.7  +MOVJ EC00074
MOVL C00075 BC00075 V=800.0  +MOVJ EC00075 VJ=100.00
MOVL C00076 BC00076 V=1000.0  +MOVJ EC00076 VJ=100.00
'EndPath S4261
'Path S4262
SFTOF3D
MOVJ C00077 BC00077 VJ=100.00  +MOVJ EC00077 VJ=100.00
MOVL C00078 BC00078 V=800.0  +MOVJ EC00078 VJ=100.00
SMOVL C00079 BC00079 V=166.7  +MOVJ EC00079
SREFP 3 C00080 BC00080  +REFP EC00080
CALL JOB:SEARCH-R1-S13D
SET P026 P006
SFTON3D P026
SMOVL C00081 BC00081 V=166.7  +MOVJ EC00081
SMOVL C00082 BC00082 V=166.7  +MOVJ EC00082
SREFP 3 C00083 BC00083  +REFP EC00083
CALL JOB:SEARCH-R1-S13D
SET P026 P006
SFTON3D P026
SMOVL C00084 BC00084 V=166.7  +MOVJ EC00084
SMOVL C00085 BC00085 V=166.7  +MOVJ EC00085
SMOVL C00086 BC00086 V=166.7  +MOVJ EC00086
SREFP 3 C00087 BC00087  +REFP EC00087
CALL JOB:SEARCH-R1-S13D
SET P026 P006
SFTON3D P026
SMOVL C00088 BC00088 V=166.7  +MOVJ EC00088
SMOVL C00089 BC00089 V=166.7  +MOVJ EC00089
SMOVL C00090 BC00090 V=166.7  +MOVJ EC00090
MOVL C00091 BC00091 V=800.0  +MOVJ EC00091 VJ=100.00
MOVL C00092 BC00092 V=1000.0  +MOVJ EC00092 VJ=100.00
'EndPath S4262
'Path S4263
SFTOF3D
MOVJ C00093 BC00093 VJ=100.00  +MOVJ EC00093 VJ=100.00
MOVL C00094 BC00094 V=800.0  +MOVJ EC00094 VJ=100.00
SMOVL C00095 BC00095 V=166.7  +MOVJ EC00095
SREFP 3 C00096 BC00096  +REFP EC00096
CALL JOB:SEARCH-R1-S13D
SET P027 P006
SFTON3D P027
SMOVL C00097 BC00097 V=166.7  +MOVJ EC00097
SMOVL C00098 BC00098 V=166.7  +MOVJ EC00098
SREFP 3 C00099 BC00099  +REFP EC00099
CALL JOB:SEARCH-R1-S13D
SET P027 P006
SFTON3D P027
SMOVL C00100 BC00100 V=166.7  +MOVJ EC00100
SMOVL C00101 BC00101 V=166.7  +MOVJ EC00101
SMOVL C00102 BC00102 V=166.7  +MOVJ EC00102
SREFP 3 C00103 BC00103  +REFP EC00103
CALL JOB:SEARCH-R1-S13D
SET P027 P006
SFTON3D P027
SMOVL C00104 BC00104 V=166.7  +MOVJ EC00104
SMOVL C00105 BC00105 V=166.7  +MOVJ EC00105
SMOVL C00106 BC00106 V=166.7  +MOVJ EC00106
MOVL C00107 BC00107 V=800.0  +MOVJ EC00107 VJ=100.00
MOVL C00108 BC00108 V=1000.0  +MOVJ EC00108 VJ=100.00
'EndPath S4263
'
'Path W4264
SFTOF3D
SFTON3D P027
MOVJ C00109 BC00109 VJ=100.00  +MOVJ EC00109 VJ=100.00
MOVJ C00110 BC00110 VJ=100.00  +MOVJ EC00110 VJ=100.00
SMOVL C00111 BC00111 V=800.0  +MOVJ EC00111
SMOVL C00112 BC00112 V=150.0 PL=0  +MOVJ EC00112
MACRO1 MJ#(0) ARGF9
ARCON
SMOVL C00113 BC00113 V=10.0  +MOVJ EC00113
SMOVL C00114 BC00114 V=10.0  +MOVJ EC00114
SMOVL C00115 BC00115 V=7.5  +MOVJ EC00115
SMOVL C00116 BC00116 V=10.0  +MOVJ EC00116
ARCOF
SMOVL C00117 BC00117 V=800.0  +MOVJ EC00117
SMOVL C00118 BC00118 V=1000.0  +MOVJ EC00118
SFTOF3D
'EndPath W4264
MOVJ C00119 BC00119 VJ=100.00  +MOVJ EC00119 VJ=100.00
MOVJ C00120 BC00120 VJ=100.00  +MOVJ EC00120 VJ=100.00
MOVJ C00121 BC00121 VJ=100.00  +MOVJ EC00121 VJ=100.00
'Path W4265
SFTOF3D
SFTON3D P021
MOVJ C00122 BC00122 VJ=100.00  +MOVJ EC00122 VJ=100.00
SMOVL C00123 BC00123 V=800.0  +MOVJ EC00123
SMOVL C00124 BC00124 V=150.0 PL=0  +MOVJ EC00124
ARCON
SMOVL C00125 BC00125 V=10.0  +MOVJ EC00125
SMOVL C00126 BC00126 V=7.5  +MOVJ EC00126
SMOVL C00127 BC00127 V=7.5  +MOVJ EC00127
SFTON3D P031
SMOVL C00128 BC00128 V=9.2  +MOVJ EC00128
SMOVL C00129 BC00129 V=9.2  +MOVJ EC00129
ARCOF
SMOVL C00130 BC00130 V=250.0  +MOVJ EC00130
SMOVL C00131 BC00131 V=800.0  +MOVJ EC00131
SMOVL C00132 BC00132 V=1000.0  +MOVJ EC00132
SFTOF3D
'EndPath W4265
MOVJ C00133 BC00133 VJ=100.00  +MOVJ EC00133 VJ=100.00
MOVJ C00134 BC00134 VJ=100.00  +MOVJ EC00134 VJ=100.00
MOVJ C00135 BC00135 VJ=100.00  +MOVJ EC00135 VJ=100.00
'Path W4266
SFTOF3D
SFTON3D P025
MOVJ C00136 BC00136 VJ=100.00  +MOVJ EC00136 VJ=100.00
SMOVL C00137 BC00137 V=800.0  +MOVJ EC00137
SMOVL C00138 BC00138 V=150.0 PL=0  +MOVJ EC00138
ARCON
SMOVL C00139 BC00139 V=9.2  +MOVJ EC00139
SMOVL C00140 BC00140 V=9.2  +MOVJ EC00140
SMOVL C00141 BC00141 V=10.0  +MOVJ EC00141
SMOVL C00142 BC00142 V=9.2  +MOVJ EC00142
SMOVL C00143 BC00143 V=9.2  +MOVJ EC00143
SMOVL C00144 BC00144 V=9.2  +MOVJ EC00144
ARCOF
SMOVL C00145 BC00145 V=800.0  +MOVJ EC00145
SMOVL C00146 BC00146 V=1000.0  +MOVJ EC00146
SFTOF3D
'EndPath W4266
MOVJ C00147 BC00147 VJ=100.00  +MOVJ EC00147 VJ=100.00
MOVJ C00148 BC00148 VJ=100.00  +MOVJ EC00148 VJ=100.00
MOVJ C00149 BC00149 VJ=100.00  +MOVJ EC00149 VJ=100.00
'Path W4267
SFTOF3D
SFTON3D P023
MOVJ C00150 BC00150 VJ=100.00  +MOVJ EC00150 VJ=100.00
SMOVL C00151 BC00151 V=800.0  +MOVJ EC00151
SMOVL C00152 BC00152 V=150.0 PL=0  +MOVJ EC00152
ARCON
SMOVL C00153 BC00153 V=9.2  +MOVJ EC00153
SMOVL C00154 BC00154 V=9.2  +MOVJ EC00154
SMOVL C00155 BC00155 V=9.2  +MOVJ EC00155
SMOVL C00156 BC00156 V=9.2  +MOVJ EC00156
SMOVL C00157 BC00157 V=9.2  +MOVJ EC00157
SMOVL C00158 BC00158 V=9.2  +MOVJ EC00158
ARCOF
SMOVL C00159 BC00159 V=800.0  +MOVJ EC00159
SMOVL C00160 BC00160 V=1000.0  +MOVJ EC00160
SFTOF3D
'EndPath W4267
MOVJ C00161 BC00161 VJ=100.00  +MOVJ EC00161 VJ=100.00
MOVJ C00162 BC00162 VJ=100.00  +MOVJ EC00162 VJ=100.00
'
'Path W4268
SFTOF3D
SFTON3D P026
MOVJ C00163 BC00163 VJ=100.00  +MOVJ EC00163 VJ=100.00
SMOVL C00164 BC00164 V=800.0  +MOVJ EC00164
SMOVL C00165 BC00165 V=150.0 PL=0  +MOVJ EC00165
ARCON
SMOVL C00166 BC00166 V=9.2  +MOVJ EC00166
SMOVL C00167 BC00167 V=9.2  +MOVJ EC00167
SMOVL C00168 BC00168 V=9.2  +MOVJ EC00168
SMOVL C00169 BC00169 V=9.2  +MOVJ EC00169
ARCOF
SMOVL C00170 BC00170 V=800.0  +MOVJ EC00170
SMOVL C00171 BC00171 V=1000.0  +MOVJ EC00171
SFTOF3D
'EndPath W4268
MOVJ C00172 BC00172 VJ=100.00  +MOVJ EC00172 VJ=100.00
MOVJ C00173 BC00173 VJ=100.00  +MOVJ EC00173 VJ=100.00
MOVJ C00174 BC00174 VJ=100.00  +MOVJ EC00174 VJ=100.00
'Path W3636
SFTOF3D
SFTON3D P022
MOVJ C00175 BC00175 VJ=100.00  +MOVJ EC00175 VJ=100.00
SMOVL C00176 BC00176 V=800.0  +MOVJ EC00176
SMOVL C00177 BC00177 V=150.0 PL=0  +MOVJ EC00177
ARCON
SMOVL C00178 BC00178 V=9.2  +MOVJ EC00178
SMOVL C00179 BC00179 V=9.2  +MOVJ EC00179
SMOVL C00180 BC00180 V=9.2  +MOVJ EC00180
SMOVL C00181 BC00181 V=9.2  +MOVJ EC00181
SMOVL C00182 BC00182 V=9.2  +MOVJ EC00182
SMOVL C00183 BC00183 V=9.2  +MOVJ EC00183
ARCOF
SMOVL C00184 BC00184 V=800.0  +MOVJ EC00184
SMOVL C00185 BC00185 V=1000.0  +MOVJ EC00185
SFTOF3D
'EndPath W3636
'Path W4269
SFTOF3D
SFTON3D P024
MOVJ C00186 BC00186 VJ=100.00  +MOVJ EC00186 VJ=100.00
SMOVL C00187 BC00187 V=800.0  +MOVJ EC00187
SMOVL C00188 BC00188 V=150.0 PL=0  +MOVJ EC00188
ARCON
SMOVL C00189 BC00189 V=9.2  +MOVJ EC00189
SMOVL C00190 BC00190 V=9.2  +MOVJ EC00190
SMOVL C00191 BC00191 V=9.2  +MOVJ EC00191
SMOVL C00192 BC00192 V=9.2  +MOVJ EC00192
SMOVL C00193 BC00193 V=9.2  +MOVJ EC00193
SMOVL C00194 BC00194 V=9.2  +MOVJ EC00194
ARCOF
SMOVL C00195 BC00195 V=800.0  +MOVJ EC00195
SMOVL C00196 BC00196 V=1000.0  +MOVJ EC00196
SFTOF3D
'EndPath W4269
MOVJ C00197 BC00197 VJ=100.00  +MOVJ EC00197 VJ=100.00
MOVJ C00198 BC00198 VJ=100.00  +MOVJ EC00198 VJ=100.00
MOVJ C00199 BC00199 VJ=100.00  +MOVJ EC00199 VJ=100.00
CALL JOB:CLEAN-R1_KM_NEW
'
'
'
'Cut-Wire
MOVJ C00200 BC00200 VJ=100.00  +MOVJ EC00200 VJ=100.00
MOVJ C00201 BC00201 VJ=100.00  +MOVJ EC00201 VJ=100.00
MOVJ C00202 BC00202 VJ=100.00  +MOVJ EC00202 VJ=100.00
'obrot
MOVJ C00203 BC00203 VJ=100.00  +MOVJ EC00203 VJ=100.00
MOVJ C00204 BC00204 VJ=100.00  +MOVJ EC00204 VJ=100.00
MOVJ C00205 BC00205 VJ=100.00  +MOVJ EC00205 VJ=100.00
'Path S4271
SFTOF3D
MOVJ C00206 BC00206 VJ=100.00  +MOVJ EC00206 VJ=100.00
MOVL C00207 BC00207 V=800.0  +MOVJ EC00207 VJ=100.00
SMOVL C00208 BC00208 V=166.7  +MOVJ EC00208
SREFP 3 C00209 BC00209  +REFP EC00209
CALL JOB:SEARCH-R1-S13D
SET P021 P006
SFTON3D P021
SMOVL C00210 BC00210 V=166.7  +MOVJ EC00210
SREFP 3 C00211 BC00211  +REFP EC00211
CALL JOB:SEARCH-R1-S13D
SET P021 P006
SFTON3D P021
SMOVL C00212 BC00212 V=166.7  +MOVJ EC00212
'EndPath S4271
'Path S4272
SFTOF3D
MOVJ C00213 BC00213 VJ=100.00  +MOVJ EC00213 VJ=100.00
SMOVL C00214 BC00214 V=166.7  +MOVJ EC00214
SREFP 3 C00215 BC00215  +REFP EC00215
CALL JOB:SEARCH-R1-S13D
SET P022 P006
SFTON3D P022
SMOVL C00216 BC00216 V=166.7  +MOVJ EC00216
SMOVL C00217 BC00217 V=166.7  +MOVJ EC00217
SREFP 3 C00218 BC00218  +REFP EC00218
CALL JOB:SEARCH-R1-S13D
SET P022 P006
SFTON3D P022
SMOVL C00219 BC00219 V=166.7  +MOVJ EC00219
SMOVL C00220 BC00220 V=166.7  +MOVJ EC00220
SMOVL C00221 BC00221 V=166.7  +MOVJ EC00221
SREFP 3 C00222 BC00222  +REFP EC00222
CALL JOB:SEARCH-R1-S13D
SET P022 P006
SFTON3D P022
SMOVL C00223 BC00223 V=166.7  +MOVJ EC00223
'EndPath S4272
'Path S4273
SFTOF3D
MOVL C00224 BC00224 V=800.0  +MOVJ EC00224 VJ=100.00
SMOVL C00225 BC00225 V=166.7  +MOVJ EC00225
SREFP 3 C00226 BC00226  +REFP EC00226
CALL JOB:SEARCH-R1-S13D
SET P023 P006
SFTON3D P023
SMOVL C00227 BC00227 V=166.7  +MOVJ EC00227
SREFP 3 C00228 BC00228  +REFP EC00228
CALL JOB:SEARCH-R1-S13D
SET P023 P006
SFTON3D P023
SMOVL C00229 BC00229 V=166.7  +MOVJ EC00229
SMOVL C00230 BC00230 V=166.7  +MOVJ EC00230
SREFP 3 C00231 BC00231  +REFP EC00231
CALL JOB:SEARCH-R1-S13D
SET P023 P006
SFTON3D P023
SMOVL C00232 BC00232 V=166.7  +MOVJ EC00232
MOVL C00233 BC00233 V=1000.0  +MOVJ EC00233 VJ=100.00
'EndPath S4273
'Path S4274
SFTOF3D
MOVJ C00234 BC00234 VJ=100.00  +MOVJ EC00234 VJ=100.00
SMOVL C00235 BC00235 V=166.7  +MOVJ EC00235
SREFP 3 C00236 BC00236  +REFP EC00236
CALL JOB:SEARCH-R1-S13D
SET P024 P006
SFTON3D P024
SMOVL C00237 BC00237 V=166.7  +MOVJ EC00237
SREFP 3 C00238 BC00238  +REFP EC00238
CALL JOB:SEARCH-R1-S13D
SET P024 P006
SFTON3D P024
SMOVL C00239 BC00239 V=166.7  +MOVJ EC00239
SMOVL C00240 BC00240 V=166.7  +MOVJ EC00240
SMOVL C00241 BC00241 V=166.7  +MOVJ EC00241
SREFP 3 C00242 BC00242  +REFP EC00242
CALL JOB:SEARCH-R1-S13D
SET P024 P006
SFTON3D P024
SMOVL C00243 BC00243 V=166.7  +MOVJ EC00243
'EndPath S4274
'Path S4275
SFTOF3D
MOVL C00244 BC00244 V=800.0  +MOVJ EC00244 VJ=100.00
SMOVL C00245 BC00245 V=166.7  +MOVJ EC00245
SREFP 3 C00246 BC00246  +REFP EC00246
CALL JOB:SEARCH-R1-S13D
SET P025 P006
SFTON3D P025
SMOVL C00247 BC00247 V=166.7  +MOVJ EC00247
SMOVL C00248 BC00248 V=166.7  +MOVJ EC00248
SREFP 3 C00249 BC00249  +REFP EC00249
CALL JOB:SEARCH-R1-S13D
SET P025 P006
SFTON3D P025
SMOVL C00250 BC00250 V=166.7  +MOVJ EC00250
SMOVL C00251 BC00251 V=166.7  +MOVJ EC00251
SREFP 3 C00252 BC00252  +REFP EC00252
CALL JOB:SEARCH-R1-S13D
SET P025 P006
SFTON3D P025
SMOVL C00253 BC00253 V=166.7  +MOVJ EC00253
SFTOF3D
SMOVL C00254 BC00254 V=250.0  +MOVJ EC00254
SREFP 3 C00255 BC00255  +REFP EC00255
CALL JOB:SEARCH-R1-S13D
SET P026 P006
SFTON3D P026
SMOVL C00256 BC00256 V=166.7  +MOVJ EC00256
SREFP 3 C00257 BC00257  +REFP EC00257
CALL JOB:SEARCH-R1-S13D
SET P026 P006
SFTON3D P026
SMOVL C00258 BC00258 V=166.7  +MOVJ EC00258
SMOVL C00259 BC00259 V=250.0  +MOVJ EC00259
SMOVL C00260 BC00260 V=166.7  +MOVJ EC00260
SREFP 3 C00261 BC00261  +REFP EC00261
CALL JOB:SEARCH-R1-S13D
SET P026 P006
SFTON3D P026
SMOVL C00262 BC00262 V=166.7  +MOVJ EC00262
'EndPath S4276
'Path S4277
SFTOF3D
MOVL C00263 BC00263 V=800.0  +MOVJ EC00263 VJ=100.00
SMOVL C00264 BC00264 V=166.7  +MOVJ EC00264
SREFP 3 C00265 BC00265  +REFP EC00265
CALL JOB:SEARCH-R1-S13D
SET P027 P006
SFTON3D P027
SMOVL C00266 BC00266 V=166.7  +MOVJ EC00266
SMOVL C00267 BC00267 V=166.7  +MOVJ EC00267
SREFP 3 C00268 BC00268  +REFP EC00268
CALL JOB:SEARCH-R1-S13D
SET P027 P006
SFTON3D P027
SMOVL C00269 BC00269 V=166.7  +MOVJ EC00269
SMOVL C00270 BC00270 V=166.7  +MOVJ EC00270
SMOVL C00271 BC00271 V=166.7  +MOVJ EC00271
SREFP 3 C00272 BC00272  +REFP EC00272
CALL JOB:SEARCH-R1-S13D
SET P027 P006
SFTON3D P027
SMOVL C00273 BC00273 V=166.7  +MOVJ EC00273
SMOVL C00274 BC00274 V=166.7  +MOVJ EC00274
SMOVL C00275 BC00275 V=166.7  +MOVJ EC00275
MOVL C00276 BC00276 V=800.0  +MOVJ EC00276 VJ=100.00
MOVL C00277 BC00277 V=500.0  +MOVJ EC00277 VJ=100.00
'EndPath S4277
'
'Path W4278
SFTOF3D
SFTON3D P027
MOVJ C00278 BC00278 VJ=40.00  +MOVJ EC00278 VJ=100.00
SMOVL C00279 BC00279 V=800.0  +MOVJ EC00279
SMOVL C00280 BC00280 V=150.0 PL=0  +MOVJ EC00280
ARCON
SMOVL C00281 BC00281 V=10.0  +MOVJ EC00281
SMOVL C00282 BC00282 V=10.0  +MOVJ EC00282
ARCOF
SMOVL C00283 BC00283 V=800.0  +MOVJ EC00283
SMOVL C00284 BC00284 V=1000.0  +MOVJ EC00284
SFTOF3D
'EndPath W4278
MOVJ C00285 BC00285 VJ=100.00  +MOVJ EC00285 VJ=100.00
MOVJ C00286 BC00286 VJ=100.00  +MOVJ EC00286 VJ=100.00
MOVJ C00287 BC00287 VJ=100.00  +MOVJ EC00287 VJ=100.00
'Path W4279
SFTOF3D
SFTON3D P021
MOVJ C00288 BC00288 VJ=100.00  +MOVJ EC00288 VJ=100.00
SMOVL C00289 BC00289 V=800.0  +MOVJ EC00289
SMOVL C00290 BC00290 V=150.0 PL=0  +MOVJ EC00290
SMOVL C00291 BC00291 V=10.0  +MOVJ EC00291
SMOVL C00292 BC00292 V=10.0  +MOVJ EC00292
SMOVL C00293 BC00293 V=10.0  +MOVJ EC00293
ARCOF
SMOVL C00294 BC00294 V=800.0  +MOVJ EC00294
SMOVL C00295 BC00295 V=1000.0  +MOVJ EC00295
SFTOF3D
'EndPath W4279
MOVJ C00296 BC00296 VJ=100.00  +MOVJ EC00296 VJ=100.00
SMOVL C00297 BC00297 V=500.0  +MOVJ EC00297
'Path W4280
SFTOF3D
SFTON3D P025
SMOVL C00298 BC00298 V=800.0  +MOVJ EC00298
SMOVL C00299 BC00299 V=150.0 PL=0  +MOVJ EC00299
ARCON
SMOVL C00300 BC00300 V=10.0  +MOVJ EC00300
SMOVL C00301 BC00301 V=10.0  +MOVJ EC00301
SMOVL C00302 BC00302 V=10.0  +MOVJ EC00302
SMOVL C00303 BC00303 V=10.0  +MOVJ EC00303
SMOVL C00304 BC00304 V=10.0  +MOVJ EC00304
SMOVL C00305 BC00305 V=10.0  +MOVJ EC00305
ARCOF
SMOVL C00306 BC00306 V=800.0  +MOVJ EC00306
SMOVL C00307 BC00307 V=1000.0  +MOVJ EC00307
SFTOF3D
'EndPath W4280
MOVJ C00308 BC00308 VJ=100.00  +MOVJ EC00308 VJ=100.00
'Path W4281
SFTOF3D
SFTON3D P023
MOVJ C00309 BC00309 VJ=100.00  +MOVJ EC00309 VJ=100.00
SMOVL C00310 BC00310 V=800.0  +MOVJ EC00310
SMOVL C00311 BC00311 V=150.0 PL=0  +MOVJ EC00311
ARCON
SMOVL C00312 BC00312 V=10.0  +MOVJ EC00312
SMOVL C00313 BC00313 V=10.0  +MOVJ EC00313
SMOVL C00314 BC00314 V=10.0  +MOVJ EC00314
SMOVL C00315 BC00315 V=10.0  +MOVJ EC00315
SMOVL C00316 BC00316 V=10.0  +MOVJ EC00316
SMOVL C00317 BC00317 V=10.0  +MOVJ EC00317
ARCOF
SMOVL C00318 BC00318 V=800.0  +MOVJ EC00318
SMOVL C00319 BC00319 V=1000.0  +MOVJ EC00319
SFTOF3D
'EndPath W4281
MOVJ C00320 BC00320 VJ=100.00  +MOVJ EC00320 VJ=100.00
'
'Path W4282
SFTOF3D
SFTON3D P026
MOVJ C00321 BC00321 VJ=100.00  +MOVJ EC00321 VJ=100.00
SMOVL C00322 BC00322 V=800.0  +MOVJ EC00322
SMOVL C00323 BC00323 V=150.0 PL=0  +MOVJ EC00323
ARCON
SMOVL C00324 BC00324 V=10.0  +MOVJ EC00324
SMOVL C00325 BC00325 V=10.0  +MOVJ EC00325
SMOVL C00326 BC00326 V=10.0  +MOVJ EC00326
SMOVL C00327 BC00327 V=10.0  +MOVJ EC00327
ARCOF
SMOVL C00328 BC00328 V=800.0  +MOVJ EC00328
SMOVL C00329 BC00329 V=1000.0  +MOVJ EC00329
SFTOF3D
'EndPath W4282
MOVJ C00330 BC00330 VJ=100.00  +MOVJ EC00330 VJ=100.00
MOVJ C00331 BC00331 VJ=100.00  +MOVJ EC00331 VJ=100.00
MOVJ C00332 BC00332 VJ=100.00  +MOVJ EC00332 VJ=100.00
'Path W4283
SFTOF3D
SFTON3D P022
MOVJ C00333 BC00333 VJ=100.00  +MOVJ EC00333 VJ=100.00
SMOVL C00334 BC00334 V=800.0  +MOVJ EC00334
SMOVL C00335 BC00335 V=150.0 PL=0  +MOVJ EC00335
ARCON
SMOVL C00336 BC00336 V=10.0  +MOVJ EC00336
SMOVL C00337 BC00337 V=10.0  +MOVJ EC00337
SMOVL C00338 BC00338 V=10.0  +MOVJ EC00338
SMOVL C00339 BC00339 V=10.0  +MOVJ EC00339
SMOVL C00340 BC00340 V=10.0  +MOVJ EC00340
SMOVL C00341 BC00341 V=10.0  +MOVJ EC00341
ARCOF
SMOVL C00342 BC00342 V=800.0  +MOVJ EC00342
SMOVL C00343 BC00343 V=1000.0  +MOVJ EC00343
SFTOF3D
'EndPath W4283
'Path W4284
SFTOF3D
SFTON3D P024
MOVJ C00344 BC00344 VJ=100.00  +MOVJ EC00344 VJ=100.00
SMOVL C00345 BC00345 V=800.0  +MOVJ EC00345
SMOVL C00346 BC00346 V=150.0 PL=0  +MOVJ EC00346
ARCON
SMOVL C00347 BC00347 V=10.0  +MOVJ EC00347
SMOVL C00348 BC00348 V=10.0  +MOVJ EC00348
SMOVL C00349 BC00349 V=10.0  +MOVJ EC00349
SMOVL C00350 BC00350 V=10.0  +MOVJ EC00350
SMOVL C00351 BC00351 V=10.0  +MOVJ EC00351
SMOVL C00352 BC00352 V=10.0  +MOVJ EC00352
ARCOF
SMOVL C00353 BC00353 V=800.0  +MOVJ EC00353
SMOVL C00354 BC00354 V=1000.0  +MOVJ EC00354
SFTOF3D
'EndPath W4284
'
MOVJ C00355 BC00355 VJ=100.00  +MOVJ EC00355 VJ=100.00
MOVJ C00356 BC00356 VJ=100.00  +MOVJ EC00356 VJ=100.00
MOVJ C00357 BC00357 VJ=100.00  +MOVJ EC00357 VJ=100.00
'obrot
MOVJ C00358 BC00358 VJ=100.00  +MOVJ EC00358 VJ=100.00
MOVJ C00359 BC00359 VJ=100.00  +MOVJ EC00359 VJ=100.00
'
MOVJ C00360 BC00360 VJ=100.00  +MOVJ EC00360 VJ=100.00
'
END
